ABB RobotStudio station: EstacionTaladrado.rspag

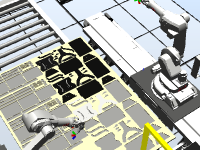
--- station ---
Station EstacionTaladrado (saved by RobotStudio 6.8.8307.1040)
Controller IRB1600APM, task T_ROB2: task frame (RAPID world) sits at (108, -1423.5, 460) mm, rotated rx 0 ry 0 rz 90 deg in the station
Controller IRB1600APM, task T_ROB1: task frame (RAPID world) sits at (108, -1423.5, 460) mm, rotated rx 0 ry 0 rz 90 deg in the station
Controller IRB1600APM
  mechanical unit ROB_1: IRB1600_6_145_A, 6 joints, base frame (0, 0, 0) mm
  mechanical unit TRACK_1: IRBT2005_IRB_STD_INT_0_0_4_A, 1 joints, base frame (0, 0, 0) mm
  mechanical unit ROB_2: IRB1600_6_145_B, 6 joints, base frame (1847, 2866, 0) mm, rotated rx 0 ry 0 rz 180 deg
  mechanical unit TRACK_2: IRBT2005_IRB_STD_INT_0_0_4_B, 1 joints, base frame (1847, 2866, 0) mm, rotated rx 0 ry 0 rz 180 deg
Layout (positions relative to the parent item):
  - Placa_de_Corte [part] at (-2250, -1220, 450) mm
  - IRC5_Singel-Cabinet [part, from Equipment\IRC5_Singel-Cabinet.rslib] at (500, 3000, 100) mm, rotated rx 90 ry 0 rz 90 deg
  - 1320_4000_h2 [part, from Equipment\Conveyor 1320 4000 h2.rslib] at (-1985, 2800, 0) mm, rotated rx 0 ry 0 rz -90 deg
  - Ventosa_Smart [smart component]
      signals: DI StartAttacher, DO Executed
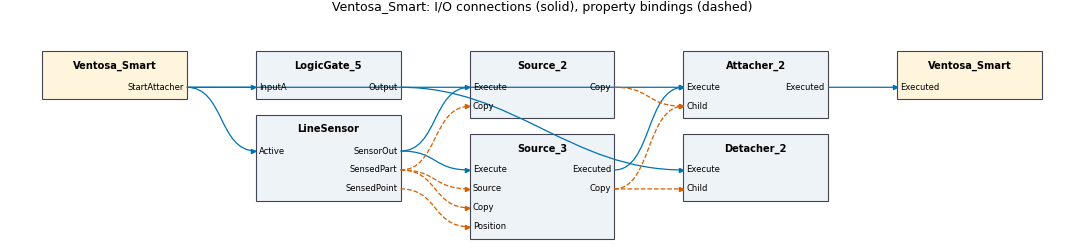
      connections:
        Ventosa_Smart.StartAttacher -> LogicGate_5.InputA
        LogicGate_5.Output -> Detacher_2.Execute
        Ventosa_Smart.StartAttacher -> LineSensor.Active
        Ventosa_Smart.StartAttacher -> Attacher_2.Execute
        Attacher_2.Executed -> Ventosa_Smart.Executed
        LineSensor.SensorOut -> Source_2.Execute
        LineSensor.SensorOut -> Source_3.Execute
        Source_3.Executed -> Attacher_2.Execute
        LineSensor.SensedPart => Source_2.Copy
        Source_2.Copy => Attacher_2.Child
        LineSensor.SensedPart => Source_3.Source
        LineSensor.SensedPart => Source_3.Copy
        Source_3.Copy => Attacher_2.Child
        Source_3.Copy => Detacher_2.Child
        LineSensor.SensedPoint => Source_3.Position
    - Attacher_2 [smart component, from Components\Attacher.rslib]
        properties: Parent=Ventosa; Flange=0; Child=(none); Mount=false; Offset=[0 0 0]; Orientation=[0 0 0]
    - Detacher_2 [smart component, from Components\Detacher.rslib]
        properties: Child=(none); KeepPosition=true
    - LogicGate_5 [smart component, from Components\LogicGate.rslib]
        properties: Operator=NOT; Delay=0
    - LineSensor [smart component, from Components\LineSensor.rslib] at (108, 403.05, 1559) mm, rotated rx 180 ry 60 rz -90 deg
        properties: Start=[0 0 0]; End=[6.66133814775094E-16 -4.71844785465692E-16 0.00999998807907376]; Radius=0.006; SensedPart=(none); SensedPoint=[0 0 0]
      - _sensorPart_ [part]
    - Ventosa [mechanism, from Libraries\Ventosa.rslib] at (108, 307.79, 1614) mm, rotated rx 180 ry 60 rz -90 deg
    - Source_3 [smart component, from Components\Source.rslib]
        properties: Source=(none); Copy=(none); Parent=(none); Position=[0 0 0]; Orientation=[0 0 0]; Transient=false; PhysicsBehavior=0
  - PLACA_SOPORTE_1 [part] at (-1200.46, 988.98, 450) mm
  - BANDEJA_LAMINA [part]
  - MyTool [mechanism, from Training Objects\myTool.rslib] at (-1542.16, -501.5, 845.83) mm, rotated rx 180 ry 0 rz 180 deg
  - SOPORTE_LATERAL_SOPORTE_1 [part] at (-961.81, 1075.54, 450) mm
  - MESA_TALADRADO [part] at (1200, -500, 400) mm
  - MESA_TALADRADO_B [part] at (-3850, -500, 400) mm
  - IRB1600_6_145_A [mechanism, from Robots\IRB1600_6_145_G_02.rslib] at (108, -498.5, 460) mm, rotated rx 0 ry 0 rz 90 deg; joint values [0, 0, 0, 0, 0.5236, 0] (rad or m)
  - IRB1600_6_145_B [mechanism, from Robots\IRB1600_6_145_G_02.rslib] at (-2758, -501.5, 460) mm, rotated rx 0 ry 0 rz -90 deg; joint values [1.5708, 1.0472, -0.3491, 0, 0.8727, 0] (rad or m)
  - IRBT2005_IRB_STD_INT_0_0_4_A [mechanism] at (400, -2248, 0) mm, rotated rx 0 ry 0 rz 90 deg; joint values [0.925] (rad or m)
      links: Base, Link1
  - IRBT2005_IRB_STD_INT_0_0_4_B [mechanism] at (-3050, 1248, 0) mm, rotated rx 0 ry 0 rz -90 deg; joint values [0.925] (rad or m)
      links: Base, Link1
  - Conveyor_A [smart component]
      signals: DI MoveConv
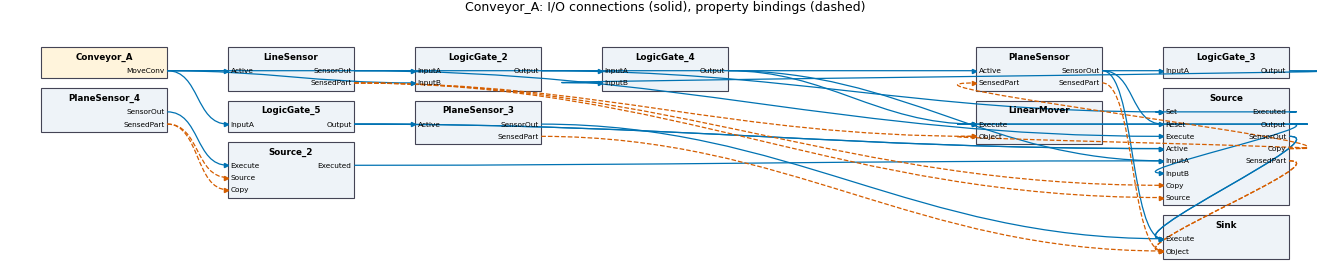
      connections:
        Source.Executed -> LogicSRLatch.Set
        PlaneSensor.SensorOut -> LogicSRLatch.Reset
        Conveyor_A.MoveConv -> LineSensor.Active
        LineSensor.SensorOut -> Source.Execute
        LogicSRLatch.Output -> LinearMover.Execute
        Conveyor_A.MoveConv -> PlaneSensor.Active
        LineSensor.SensorOut -> LogicGate_2.InputA
        Conveyor_A.MoveConv -> LogicGate_2.InputB
        LogicGate_2.Output -> LogicSRLatch.Set
        PlaneSensor.SensorOut -> LogicGate_3.InputA
        LogicGate_2.Output -> LogicGate_4.InputA
        LogicGate_3.Output -> LogicGate_4.InputB
        PlaneSensor.SensorOut -> Sink.Execute
        PlaneSensor_2.SensorOut -> Sink.Execute
        Conveyor_A.MoveConv -> LogicGate_5.InputA
        LogicGate_5.Output -> PlaneSensor_2.Active
        LogicGate_5.Output -> LineSensor.Active
        LineSensor.SensorOut -> Sink.Execute
        PlaneSensor_3.SensorOut -> Sink.Execute
        LogicGate_5.Output -> PlaneSensor_3.Active
        PlaneSensor_4.SensorOut -> Source_2.Execute
        LogicGate_4.Output -> LogicGate_8.InputA
        LogicGate_8.Output -> LinearMover.Execute
        LogicGate_9.Output -> LogicGate_8.InputB
        Source_2.Executed -> LogicGate_9.InputA
        LogicGate_4.Output -> LinearMover.Execute
        LineSensor.SensedPart => Source.Copy
        Source.Copy => LinearMover.Object
        Source.Copy => PlaneSensor.SensedPart
        LineSensor.SensedPart => Source.Source
        PlaneSensor_2.SensedPart => Sink.Object
        LineSensor.SensedPart => Sink.Object
        PlaneSensor_3.SensedPart => Sink.Object
        LineSensor.SensedPart => LinearMover.Object
        PlaneSensor.SensedPart => Sink.Object
        PlaneSensor_4.SensedPart => Source_2.Source
        PlaneSensor_4.SensedPart => Source_2.Copy
    - PlaneSensor [smart component, from Components\PlaneSensor.rslib]
        properties: Origin=[-1.025 -4.3 0.776]; Axis1=[0 0 0.099]; Axis2=[0.39 0 0]; SensedPart=(none)
      - _sensorPart_ [part]
    - LineSensor [smart component, from Components\LineSensor.rslib]
        properties: Start=[-0.83 -1.7 0.78]; End=[-0.83 -4.3 0.785]; Radius=0.005; SensedPart=BOX_A; SensedPoint=[-0.83 -1.7 0.78]
      - _sensorPart_ [part]
    - LinearMover [smart component, from Components\LinearMover.rslib]
        properties: Object=BOX_A; Direction=[0 -3.5 0]; Speed=0.5; Reference=Global; ReferenceObject=(none)
    - LogicGate_2 [smart component, from Components\LogicGate.rslib]
        properties: Operator=AND; Delay=0
    - LogicGate_3 [smart component, from Components\LogicGate.rslib]
        properties: Operator=NOT; Delay=0
    - LogicGate_4 [smart component, from Components\LogicGate.rslib]
        properties: Operator=AND; Delay=0
    - Sink [smart component, from Components\Sink.rslib]
        properties: Object=(none)
    - LogicGate_5 [smart component, from Components\LogicGate.rslib]
        properties: Operator=NOT; Delay=0
    - PlaneSensor_3 [smart component, from Components\PlaneSensor.rslib]
        properties: Origin=[-1.02 -2 0.786]; Axis1=[0.38 0 0]; Axis2=[0 0.3 0]; SensedPart=(none)
      - _sensorPart_ [part]
    - Source_2 [smart component, from Components\Source.rslib]
        properties: Source=(none); Copy=(none); Parent=(none); Position=[-0.83 -1.85 0.776]; Orientation=[0 0 0]; Transient=false; PhysicsBehavior=0
    - PlaneSensor_4 [smart component, from Components\PlaneSensor.rslib]
        properties: Origin=[-1.025 -4.3 0.776]; Axis1=[0 0 0.099]; Axis2=[0.39 0 0]; SensedPart=(none)
      - _sensorPart_ [part]
  - 400_guide_B [part, from Equipment\Conveyor Guide 400.rslib] at (-2020, -1500, 0) mm, rotated rx 0 ry 0 rz -90 deg
  - 400_guide_A [part, from Equipment\Conveyor Guide 400.rslib] at (-1030, -1500, 0) mm, rotated rx 0 ry 0 rz -90 deg
  - SOPORTE_LATERAL_SOPORTE_1_2 [part] at (-1011.44, 1038.99, 450) mm
  - BASE_SOPORTE_1 [part] at (-878.76, 996.15, 450) mm
  - GRADUADOR_INCLINACION_SOPORTE_1 [part] at (-1023.59, 997.95, 450) mm
  - GRADUADOR_INCLINACION_SOPORTE_1_2 [part] at (-966.4, 1160.33, 450) mm
  - SUJECION_CENTRAL_SOPORTE_1 [part] at (-870.47, 885.99, 450) mm
  - BRAZO_SOPORTE_1 [part] at (-762.24, 1077.84, 450) mm
  - BRAZO_2_SOPORTE_1 [part] at (-1135.46, 1150.12, 450) mm
  - BOX_A [part] at (-830, -1850, 776) mm
  - PLACA_INFERIOR_MESA_1 [part] at (-558.01, 1007.22, 450) mm
  - PLACA_SUPERIOR_MESA_1 [part] at (-913.92, 730.48, 450) mm
  - SOPORTE_LATERAL_I_MESA_1 [part] at (-1245.6, 782.8, 450) mm
  - SOPORTE_LATERAL_D_MESA_1 [part] at (-580.16, 719.3, 450) mm
  - BASE_SOPORTE_2 [part] at (-884.8, 433.69, 450) mm
  - BRAZO_2_SOPORTE_2 [part] at (-1248.93, 610.54, 450) mm
  - GRADUADOR_INCLINACION_SOPORTE_2 [part] at (-779.66, 491.03, 450) mm
  - GRADUADOR_INCLINACION_SOPORTE_2_2 [part] at (-777.34, 553.46, 450) mm
  - BRAZO_SOPORTE_3 [part] at (-1228.76, 84.41, 450) mm
  - BRAZO_SOPORTE_2 [part] at (-1242.31, 664.75, 450) mm
  - SOPORTE_LATERAL_SOPORTE_2 [part] at (-1012.51, 575.73, 450) mm
  - SOPORTE_LATERAL_SOPORTE_2_2 [part] at (-1009.84, 532.43, 450) mm
  - PLACA_SOPORTE_2 [part] at (-1204.37, 425.85, 450) mm
  - SUJECION_CENTRAL_SOPORTE_2 [part] at (-888.41, 308.37, 450) mm
  - PLACA_INFERIOR_MESA_2 [part] at (-580.45, 456.05, 450) mm
  - PLACA_SUPERIOR_MESA_2 [part] at (-915.16, 155.2, 450) mm
  - SOPORTE_LATERAL_I_MESA_2 [part] at (-1273.79, 206.85, 450) mm
  - SOPORTE_LATERAL_D_MESA_2 [part] at (-588.98, 160.74, 450) mm
  - BASE_SOPORTE_3 [part] at (-885, -169.85, 450) mm
  - PLACA_SOPORTE_3 [part] at (-1212.18, -176.73, 450) mm
  - Fence_2500 [graphiccomponentgroup, from Equipment\Fence_2500.rslib] at (-1350, -4000, 0) mm
    - Body 1 [part, from Equipment\Fence_2500.rslib]
    - Body 2 [part, from Equipment\Fence_2500.rslib]
  - Conveyor_B [smart component]
      signals: DI MoveConvB
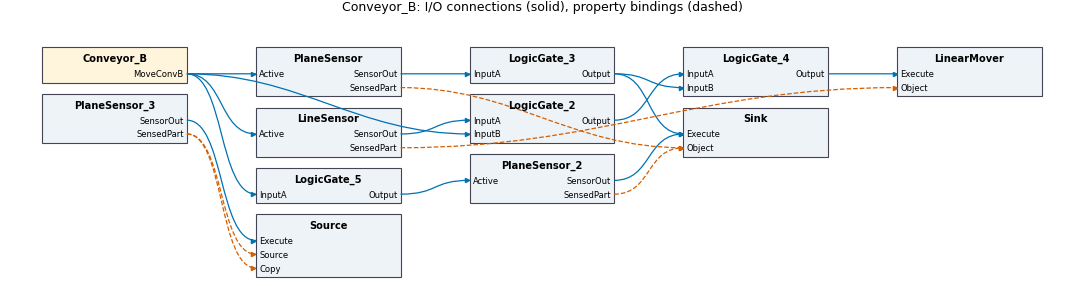
      connections:
        Conveyor_B.MoveConvB -> PlaneSensor.Active
        PlaneSensor.SensorOut -> LogicGate_3.InputA
        LogicGate_3.Output -> Sink.Execute
        Conveyor_B.MoveConvB -> LineSensor.Active
        LineSensor.SensorOut -> LogicGate_2.InputA
        Conveyor_B.MoveConvB -> LogicGate_5.InputA
        LogicGate_5.Output -> PlaneSensor_2.Active
        PlaneSensor_3.SensorOut -> Source.Execute
        LogicGate_2.Output -> LogicGate_4.InputA
        Conveyor_B.MoveConvB -> LogicGate_2.InputB
        LogicGate_3.Output -> LogicGate_4.InputB
        LogicGate_4.Output -> LinearMover.Execute
        PlaneSensor_2.SensorOut -> Sink.Execute
        PlaneSensor.SensedPart => Sink.Object
        LineSensor.SensedPart => LinearMover.Object
        PlaneSensor_3.SensedPart => Source.Source
        PlaneSensor_3.SensedPart => Source.Copy
        PlaneSensor_2.SensedPart => Sink.Object
    - LinearMover [smart component, from Components\LinearMover.rslib]
        properties: Object=BOX_A; Direction=[0 -3.5 0]; Speed=0.5; Reference=Global; ReferenceObject=(none)
    - LineSensor [smart component, from Components\LineSensor.rslib]
        properties: Start=[-1.82 -1.7 0.78]; End=[-1.82 -4.3 0.785]; Radius=0.005; SensedPart=BOX_A; SensedPoint=[-0.83 -1.7 0.78]
      - _sensorPart_ [part]
    - PlaneSensor [smart component, from Components\PlaneSensor.rslib]
        properties: Origin=[-2.02 -4.3 0.776]; Axis1=[0 0 0.099]; Axis2=[0.39 0 0]; SensedPart=(none)
      - _sensorPart_ [part]
    - PlaneSensor_2 [smart component, from Components\PlaneSensor.rslib]
        properties: Origin=[-2.01 -2 0.786]; Axis1=[0.38 0 0]; Axis2=[0 0.3 0]; SensedPart=(none)
      - _sensorPart_ [part]
    - PlaneSensor_3 [smart component, from Components\PlaneSensor.rslib]
        properties: Origin=[-2.02 -4.3 0.776]; Axis1=[0 0 0.099]; Axis2=[0.39 0 0]; SensedPart=(none)
      - _sensorPart_ [part]
    - Sink [smart component, from Components\Sink.rslib]
        properties: Object=(none)
    - Source [smart component, from Components\Source.rslib]
        properties: Source=(none); Copy=(none); Parent=(none); Position=[-0.83 -1.85 0.776]; Orientation=[0 0 0]; Transient=false; PhysicsBehavior=0
    - LogicGate_2 [smart component, from Components\LogicGate.rslib]
        properties: Operator=AND; Delay=0
    - LogicGate_3 [smart component, from Components\LogicGate.rslib]
        properties: Operator=NOT; Delay=0
    - LogicGate_4 [smart component, from Components\LogicGate.rslib]
        properties: Operator=AND; Delay=0
    - LogicGate_5 [smart component, from Components\LogicGate.rslib]
        properties: Operator=NOT; Delay=0
  - BOX_B [part] at (-1820, -1850, 776) mm
Attachment: LineSensor is attached to Ventosa / HERRAMIENTA
Attachment: Ventosa is attached to IRB1600_6_145_A / Link6
Attachment: MyTool is attached to IRB1600_6_145_B / Link6
Attachment: IRB1600_6_145_A is attached to IRBT2005_IRB_STD_INT_0_0_4_A / Link1
Attachment: IRB1600_6_145_B is attached to IRBT2005_IRB_STD_INT_0_0_4_B / Link1
Station logic (signal -> signal, property => property):
  Attacher.Executed -> LogicGate.InputB
  IRB1600APM.DOATTCH -> Ventosa_Smart.StartAttacher
  IRB1600APMSYS.DO_ATTCH_A -> Ventosa_Smart.StartAttacher
  IRB1600APM.ATTACH -> Ventosa_Smart.StartAttacher
  IRB1600APM.MoveConv -> Conveyor_A.MoveConv

--- Backups/IRB1600APM/RAPID/TASK1/PROGMOD/CalibData.mod ---
MODULE CalibData
	PERS tooldata VentosaTCP:=[TRUE,[[0,0,110.772],[1,0,0,0]],[1,[0,0,53.582],[1,0,0,0],0,0,0]];
	TASK PERS wobjdata PLACA_A:=[FALSE,TRUE,"",[[0,0,0],[1,0,0,0]],[[203.5,2358,-10],[0.707106781,0,0,-0.707106781]]];
ENDMODULE

--- Backups/IRB1600APM/RAPID/TASK1/PROGMOD/Module1.mod ---
MODULE Module1
    CONST jointtarget HOME_A:=[[0,0,0,0,30,0],[925,9E+09,9E+09,9E+09,9E+09,9E+09]];
    CONST jointtarget MID_A:=[[90,60,-20,0,50,0],[925,9E+09,9E+09,9E+09,9E+09,9E+09]];
    CONST jointtarget PS1_A:=[[87.22,84.052,-44.6,0,50.548,0],[2349.769019747,9E+09,9E+09,9E+09,9E+09,9E+09]];
    CONST jointtarget CONVEYOR_A:=[[84.914,41.92,15.328,-0.622,32.813,0],[-461.181385797,9E+09,9E+09,9E+09,9E+09,9E+09]];
    CONST jointtarget SLS1_A:=[[82.069,70.996,-7.558,0,26.562,-7.931],[2350,9E+09,9E+09,9E+09,9E+09,9E+09]];
    CONST jointtarget TABLE_A:=[[-90,71.536,-9.408,0,27.873,0],[925,9E+09,9E+09,9E+09,9E+09,9E+09]];
    CONST jointtarget PS1_AA:=[[87.22,83.446,-44.115,0,50.669,0],[2349.769019747,9E+09,9E+09,9E+09,9E+09,9E+09]];
    CONST jointtarget MID_CONV:=[[90,60,-40,0,70,0],[-500,9E+09,9E+09,9E+09,9E+09,9E+09]];
    CONST jointtarget MID_CONV_A:=[[89.175,20.381,4.444,0.004,65.253,0],[-480,9E+09,9E+09,9E+09,9E+09,9E+09]];
    CONST jointtarget PSLS1_AA:=[[82.069,69.527,-6.738,0,27.211,0],[2350,9E+09,9E+09,9E+09,9E+09,9E+09]];
    CONST jointtarget SLS12_AA:=[[84.262,72.054,-13.066,0,31.013,0],[2350,9E+09,9E+09,9E+09,9E+09,9E+09]];
    CONST jointtarget SLS12_A:=[[84.105,72.802,-13.543,0,30.74,-5.895],[2350,9E+09,9E+09,9E+09,9E+09,9E+09]];
    CONST jointtarget BS1_A:=[[84.635,68.196,3.223,0,18.581,0],[2350,9E+09,9E+09,9E+09,9E+09,9E+09]];
    CONST jointtarget BS1_AA:=[[84.635,67.383,3.658,0,18.96,0],[2350,9E+09,9E+09,9E+09,9E+09,9E+09]];
    CONST jointtarget GIS1_A:=[[86.51,72.86,-13.724,0,30.865,-3.49],[2350,9E+09,9E+09,9E+09,9E+09,9E+09]];
    CONST jointtarget GIS1_AA:=[[86.51,72.134,-13.296,0,31.162,0],[2350,9E+09,9E+09,9E+09,9E+09,9E+09]];
    CONST jointtarget GIS12_AA:=[[77.771,70.671,-8.671,0,28,0],[2350,9E+09,9E+09,9E+09,9E+09,9E+09]];
    CONST jointtarget GIS12_A:=[[77.79,71.449,-9.107,0,27.659,-12.21],[2350,9E+09,9E+09,9E+09,9E+09,9E+09]];
    CONST jointtarget BRS1_A:=[[80.135,66.069,14.969,0,8.962,-9.865],[2350,9E+09,9E+09,9E+09,9E+09,9E+09]];
    CONST jointtarget BRS1_AA:=[[80.135,65.237,15.395,0,9.368,0],[2350,9E+09,9E+09,9E+09,9E+09,9E+09]];
    CONST jointtarget BRS12_A:=[[79.805,80.411,-35.266,0,44.855,0],[2350,9E+09,9E+09,9E+09,9E+09,9E+09]];
    CONST jointtarget BRS12_AA:=[[79.805,79.69,-34.75,0,45.061,0],[2350,9E+09,9E+09,9E+09,9E+09,9E+09]];
    CONST jointtarget SCS1_A:=[[92.371,67.896,4.57,0,17.533,2.371],[2350,9E+09,9E+09,9E+09,9E+09,9E+09]];
    CONST jointtarget SCS1_AA:=[[92.371,67.108,4.99,0,17.903,0],[2350,9E+09,9E+09,9E+09,9E+09,9E+09]];
    CONST jointtarget PIM1_A:=[[56.022,65.432,22.991,0,1.578,-33.978],[1981.865508797,9E+09,9E+09,9E+09,9E+09,9E+09]];
    CONST jointtarget PIM1_AA:=[[56.022,64.534,23.445,0,2.021,-33.978],[1981.865508797,9E+09,9E+09,9E+09,9E+09,9E+09]];
    CONST jointtarget TABLE_AA:=[[-90,55.011,-3.204,0,38.193,0],[925,9E+09,9E+09,9E+09,9E+09,9E+09]];
    CONST jointtarget TABLE_A90:=[[-90.000002504,71.537536725,-9.40957169,0,27.872034908,90.000016165],[925.000071526,9E+09,9E+09,9E+09,9E+09,9E+09]];
    CONST jointtarget TABLE_A180:=[[-90,71.538,-9.41,0,27.872,180],[925.000071526,9E+09,9E+09,9E+09,9E+09,9E+09]];
    CONST jointtarget TABLE_A270:=[[-90,71.538,-9.41,0,27.872,270],[925.000071526,9E+09,9E+09,9E+09,9E+09,9E+09]];
    CONST jointtarget PSM1_AA:=[[80.44,68.736,-1.688,0.001,22.953,0],[1981.865508797,9E+09,9E+09,9E+09,9E+09,9E+09]];
    CONST jointtarget PSM1_A:=[[80.44,69.498,-2.107,0.001,22.609,0],[1981.865508797,9E+09,9E+09,9E+09,9E+09,9E+09]];
    CONST jointtarget SLIM1_AA:=[[80.586,90.25,-60.725,0,60.476,0],[1981.865508797,9E+09,9E+09,9E+09,9E+09,9E+09]];
    CONST jointtarget SLIM1_A:=[[80.586,91.085,-61.583,0,60.499,0],[1981.865508797,9E+09,9E+09,9E+09,9E+09,9E+09]];
    CONST jointtarget SLDM1_A:=[[76.838,65.923,31.968,-180,7.889,166.838],[1981.865508797,9E+09,9E+09,9E+09,9E+09,9E+09]];
    CONST jointtarget SLDM1_AA:=[[76.838,64.965,32.458,-180,7.42,166.838],[1981.865508797,9E+09,9E+09,9E+09,9E+09,9E+09]];
    CONST jointtarget SLS1_AA:=[[82.069,69.527,-6.738,0,27.211,0],[2350,9E+09,9E+09,9E+09,9E+09,9E+09]];
    CONST jointtarget TABLE_AA90:=[[-90,55.011,-3.204,0,38.193,90],[925,9E+09,9E+09,9E+09,9E+09,9E+09]];
    CONST jointtarget TABLE_AA180:=[[-90,55.011,-3.204,0,38.193,180],[925,9E+09,9E+09,9E+09,9E+09,9E+09]];
    CONST jointtarget TABLE_AA270:=[[-90,55.011,-3.204,0,38.193,270],[925,9E+09,9E+09,9E+09,9E+09,9E+09]];
    CONST jointtarget PS2_A:=[[92.202,84.352,-45.348,0,50.996,0],[1900.590004436,9E+09,9E+09,9E+09,9E+09,9E+09]];
    CONST jointtarget PS2_AA:=[[92.202,83.623,-44.761,0,51.138,0],[1900.590004436,9E+09,9E+09,9E+09,9E+09,9E+09]];
    CONST jointtarget BRS2_A:=[[82.088,89.838,-58.651,0,58.813,-7.912],[1900.590004436,9E+09,9E+09,9E+09,9E+09,9E+09]];
    CONST jointtarget BRS2_AA:=[[82.088,89.029,-57.86,0,58.831,-7.912],[1900.590004436,9E+09,9E+09,9E+09,9E+09,9E+09]];
    CONST jointtarget BRS22_A:=[[84.383,89.865,-58.714,0,58.849,0],[1900.590004436,9E+09,9E+09,9E+09,9E+09,9E+09]];
    CONST jointtarget BRS22_AA:=[[84.383,89.06,-57.926,0,58.866,0],[1900.590004436,9E+09,9E+09,9E+09,9E+09,9E+09]];
    CONST jointtarget BS2_A:=[[91.176,68.246,3.004,0,18.749,0],[1900.590004436,9E+09,9E+09,9E+09,9E+09,9E+09]];
    CONST jointtarget BS2_AA:=[[91.176,67.47,3.42,0,19.11,0],[1900.590004436,9E+09,9E+09,9E+09,9E+09,9E+09]];
    CONST jointtarget SLS2_A:=[[84.969,72.779,-13.468,0,30.689,-5.031],[1900.590004436,9E+09,9E+09,9E+09,9E+09,9E+09]];
    CONST jointtarget SLS2_AA:=[[84.969,72.056,-13.042,0,30.986,-5.031],[1900.590004436,9E+09,9E+09,9E+09,9E+09,9E+09]];
    CONST jointtarget SLS22_A:=[[87.166,72.539,-12.701,0,30.162,-2.834],[1900.590004436,9E+09,9E+09,9E+09,9E+09,9E+09]];
    CONST jointtarget SLS22_AA:=[[87.165999923,71.813298783,-12.275472962,-0.000004916,30.462172415,-2.833995324],[1900.590004436,9E+09,9E+09,9E+09,9E+09,9E+09]];
    CONST jointtarget GIS2_A:=[[113.168,67.339,7.247,0.002,15.415,23.166],[2350,9E+09,9E+09,9E+09,9E+09,9E+09]];
    CONST jointtarget GIS2_AA:=[[113.167997339,66.544675272,7.664479702,0.001953446,15.791846446,23.166056768],[2350,9E+09,9E+09,9E+09,9E+09,9E+09]];
    CONST jointtarget GIS22_A:=[[89.278,66.036,15.23,0,8.734,-0.722],[1900.590004436,9E+09,9E+09,9E+09,9E+09,9E+09]];
    CONST jointtarget GIS22_AA:=[[89.277996868,65.192591514,15.662153106,0,9.145254468,-0.722003182],[1900.590004436,9E+09,9E+09,9E+09,9E+09,9E+09]];
    CONST jointtarget SCS2_AA:=[[99.610427006,67.956188505,1.376250141,0.000001343,20.667561617,9.610424502],[1900.590004436,9E+09,9E+09,9E+09,9E+09,9E+09]];
    CONST jointtarget SCS2_A:=[[99.610427006,68.727863278,0.959277551,0.000002592,20.312857941,9.610423648],[1900.590004436,9E+09,9E+09,9E+09,9E+09,9E+09]];
    CONST jointtarget PIM2_AA:=[[91.561998466,65.215083327,34.070885788,-180.000005009,9.285968318,-178.437995387],[1898.318303054,9E+09,9E+09,9E+09,9E+09,9E+09]];
    CONST jointtarget PIM2_A:=[[91.562,66.191,33.57,-180,9.761,-178.438],[1898.318303054,9E+09,9E+09,9E+09,9E+09,9E+09]];
    CONST jointtarget PSM2_A:=[[107.463751193,70.721069572,-6.596925403,0,25.875854067,15.261750342],[1900.590004436,9E+09,9E+09,9E+09,9E+09,9E+09]];
    CONST jointtarget PSM2_AA:=[[107.463751193,69.981305443,-6.180146833,-0.000001709,26.198836637,15.261752049],[1900.590004436,9E+09,9E+09,9E+09,9E+09,9E+09]];
    CONST jointtarget SLIM2_AA:=[[101.065605639,97.834687105,-78.028074248,-0.000006825,70.193375987,8.863605642],[1900.590004436,9E+09,9E+09,9E+09,9E+09,9E+09]];
    CONST jointtarget SLIM2_A:=[[101.065605639,99.278479813,-80.225257312,-0.00000448,70.946766343,8.863604788],[1900.590004436,9E+09,9E+09,9E+09,9E+09,9E+09]];
    CONST jointtarget SLDM2_AA:=[[114.412894938,64.526784674,27.05293984,180.0003875,1.579731188,202.210537095],[1900.590004436,9E+09,9E+09,9E+09,9E+09,9E+09]];
    CONST jointtarget SLDM2_A:=[[114.412888108,65.445356325,26.587732241,179.999718141,2.033083713,202.211192794],[1900.590004436,9E+09,9E+09,9E+09,9E+09,9E+09]];
    !***********************************************************
    !
    ! Módulo:  Module1
    !
    ! Descripción:
    !   <Introduzca la descripción aquí>
    !
    ! Autor: sebas
    !
    ! Versión: 1.0
    !
    !***********************************************************


    !***********************************************************
    !
    ! Procedimiento Main
    !
    !   Este es el punto de entrada de su programa
    !
    !***********************************************************
    VAR intnum intparada;

    PROC main()
        !START
        CONNECT intparada WITH RutinaParada;
        iSignalDI STOPDI,1,intparada;
        SetDO MoveConv,0;
        WaitDI START,1;
        Path_HOME_A;
        Path_MID_A;
        !PLACA SOPORTE 1
        Path_PS1_AA;
        WaitTime 1;
        SetDO ATTACH,1;
        WaitDO ATTACH,1;
        Path_PS1_A;
        WaitTime 1;
        SetDO ATTACH,0;
        WaitDO ATTACH,0;
        Path_MID_CONV_A;
        Path_HOME_A;
        !SOPORTE LATERAL SOPORTE 1
        Path_SLS1_AA;
        WaitTime 1;
        SetDO ATTACH,1;
        WaitDO ATTACH,1;
        Path_SLS1_A;
        WaitDI DRILLCHECK,1;
        Path_SLS1_A_2;
        WaitTime 1;
        SetDO ATTACH,0;
        WaitDO ATTACH,0;
        Path_MID_CONV_A;
        Path_HOME_A;
        !SOPORTE LATERAL SOPORTE 1 2
        Path_SLS12_AA;
        WaitTime 1;
        SetDO ATTACH,1;
        WaitDO ATTACH,1;
        Path_SLS12_A;
        WaitDI DRILLCHECK,1;
        Path_SLS12_A_2;
        WaitTime 1;
        SetDO ATTACH,0;
        WaitDO ATTACH,0;
        Path_MID_CONV_A;
        Path_HOME_A;
        !BASE SOPORTE 1
        Path_BS1_AA;
        WaitTime 1;
        SetDO ATTACH,1;
        WaitDO ATTACH,1;
        Path_BS1_A;
        WaitTime 1;
        SetDO ATTACH,0;
        WaitDO ATTACH,0;
        Path_MID_CONV_A;
        Path_HOME_A;
        !GRADUADOR DE INCLINACION SOPORTE 1
        Path_GIS1_AA;
        WaitTime 1;
        SetDO ATTACH,1;
        WaitDO ATTACH,1;
        Path_GIS1_A;
        WaitDI DRILLCHECK,1;
        Path_GIS1_A_2;
        WaitTime 1;
        SetDO ATTACH,0;
        WaitDO ATTACH,0;
        Path_MID_CONV_A;
        Path_HOME_A;
        !GRADUADOR DE INCLINACION SOPORTE 1 2
        Path_GIS12_AA;
        WaitTime 1;
        SetDO ATTACH,1;
        WaitDO ATTACH,1;
        Path_GIS12_A;
        WaitDI DRILLCHECK,1;
        Path_GIS12_A_2;
        WaitTime 1;
        SetDO ATTACH,0;
        WaitDO ATTACH,0;
        Path_MID_CONV_A;
        Path_HOME_A;
        !BRAZO SOPORTE 1
        Path_BRS1_AA;
        WaitTime 1;
        SetDO ATTACH,1;
        WaitDO ATTACH,1;
        Path_BRS1_A;
        WaitTime 1;
        SetDO ATTACH,0;
        WaitDO ATTACH,0;
        Path_MID_CONV_A;
        Path_HOME_A;
        !BRAZO 2 SOPORTE 1
        Path_BRS12_AA;
        WaitTime 1;
        SetDO ATTACH,1;
        WaitDO ATTACH,1;
        Path_BRS12_A;
        WaitTime 1;
        SetDO ATTACH,0;
        WaitDO ATTACH,0;
        Path_MID_CONV_A;
        Path_HOME_A;
        !SUJECION CENTRAL SOPORTE 1
        Path_SCS1_AA;
        WaitTime 1;
        SetDO ATTACH,1;
        WaitDO ATTACH,1;
        Path_SCS1_A;
        WaitDI DRILLCHECK,1;
        Path_SCS1_A_2;
        WaitTime 1;
        SetDO ATTACH,0;
        WaitDO ATTACH,0;
        Path_MID_CONV_A;
        Path_HOME_A;
        !START CONVEYOR
        SetDO MoveConv,1;
        WaitTime 4.5;
        SetDO MoveConv,0;
        SetDO PAUSE,1;
        WaitDO PAUSE,0;
        !
        !MESA 1
        !
        !PLACA INFERIOR MESA 1
        Path_PIM1_AA;
        WaitTime 1;
        SetDO ATTACH,1;
        WaitDO ATTACH,1;
        Path_PIM1_A;
        WaitDI DRILLCHECK,1;
        WaitTime 1;
        Path_PIM1_A_2;
        WaitDI DRILLCHECK,1;
        WaitTime 1;
        Path_PIM1_A_3;
        WaitDI DRILLCHECK,1;
        WaitTime 1;
        Path_PIM1_A_4;
        WaitDI DRILLCHECK,1;
        WaitTime 1;
        Path_PIM1_A_5;
        WaitTime 1;
        SetDO ATTACH,0;
        WaitDO ATTACH,0;
        Path_MID_CONV_A;
        Path_HOME_A;
        !PLACA SUPERIOR MESA 1
        Path_PSM1_AA;
        WaitTime 1;
        SetDO ATTACH,1;
        WaitDO ATTACH,1;
        Path_PSM1_A;
        WaitTime 1;
        SetDO ATTACH,0;
        WaitDO ATTACH,0;
        Path_MID_CONV_A;
        Path_HOME_A;
        !SOPORTE LATERAL IZQUIERDO MESA 1
        Path_SLIM1_AA;
        WaitTime 1;
        SetDO ATTACH,1;
        WaitDO ATTACH,1;
        Path_SLIM1_A;
        WaitTime 1;
        SetDO ATTACH,0;
        WaitDO ATTACH,0;
        Path_MID_CONV_A;
        Path_HOME_A;
        !SOPORTE LATERAL DERECHO MESA 1
        Path_SLDM1_AA;
        WaitTime 1;
        SetDO ATTACH,1;
        WaitDO ATTACH,1;
        Path_SLDM1_A;
        WaitTime 1;
        SetDO ATTACH,0;
        WaitDO ATTACH,0;
        Path_MID_CONV_A;
        Path_HOME_A;
        !START CONVEYOR
        SetDO MoveConv,1;
        WaitTime 4.5;
        SetDO MoveConv,0;
        SetDO PAUSE,1;
        WaitDO PAUSE,0;
        !
        !SOPORTE 2
        !
        !PLACA SOPORTE 2
        Path_PS2_AA;
        WaitTime 1;
        SetDO ATTACH,1;
        WaitDO ATTACH,1;
        Path_PS2_A;
        WaitTime 1;
        SetDO ATTACH,0;
        WaitDO ATTACH,0;
        Path_MID_CONV_A;
        Path_HOME_A;
        !SOPORTE LATERAL SOPORTE 2
        Path_SLS2_AA;
        WaitTime 1;
        SetDO ATTACH,1;
        WaitDO ATTACH,1;
        Path_SLS2_A;
        WaitDI DRILLCHECK,1;
        Path_SLS2_A_2;
        WaitTime 1;
        SetDO ATTACH,0;
        WaitDO ATTACH,0;
        Path_MID_CONV_A;
        Path_HOME_A;
        !SOPORTE LATERAL SOPORTE 2 2
        Path_SLS22_AA;
        WaitTime 1;
        SetDO ATTACH,1;
        WaitDO ATTACH,1;
        Path_SLS22_A;
        WaitDI DRILLCHECK,1;
        Path_SLS22_A_2;
        WaitTime 1;
        SetDO ATTACH,0;
        WaitDO ATTACH,0;
        Path_MID_CONV_A;
        Path_HOME_A;
        !BASE SOPORTE 2
        Path_BS2_AA;
        WaitTime 1;
        SetDO ATTACH,1;
        WaitDO ATTACH,1;
        Path_BS2_A;
        WaitTime 1;
        SetDO ATTACH,0;
        WaitDO ATTACH,0;
        Path_MID_CONV_A;
        Path_HOME_A;
        !GRADUADOR DE INCLINACION SOPORTE 2
        Path_GIS2_AA;
        WaitTime 1;
        SetDO ATTACH,1;
        WaitDO ATTACH,1;
        Path_GIS2_A;
        WaitDI DRILLCHECK,1;
        Path_GIS2_A_2;
        WaitTime 1;
        SetDO ATTACH,0;
        WaitDO ATTACH,0;
        Path_MID_CONV_A;
        Path_HOME_A;
        !GRADUADOR DE INCLINACION SOPORTE 2 2
        Path_GIS22_AA;
        WaitTime 1;
        SetDO ATTACH,1;
        WaitDO ATTACH,1;
        Path_GIS22_A;
        WaitDI DRILLCHECK,1;
        Path_GIS22_A_2;
        WaitTime 1;
        SetDO ATTACH,0;
        WaitDO ATTACH,0;
        Path_MID_CONV_A;
        Path_HOME_A;
        !BRAZO SOPORTE 2
        Path_BRS2_AA;
        WaitTime 1;
        SetDO ATTACH,1;
        WaitDO ATTACH,1;
        Path_BRS2_A;
        WaitTime 1;
        SetDO ATTACH,0;
        WaitDO ATTACH,0;
        Path_MID_CONV_A;
        Path_HOME_A;
        !BRAZO 2 SOPORTE 2
        Path_BRS22_AA;
        WaitTime 1;
        SetDO ATTACH,1;
        WaitDO ATTACH,1;
        Path_BRS22_A;
        WaitTime 1;
        SetDO ATTACH,0;
        WaitDO ATTACH,0;
        Path_MID_CONV_A;
        Path_HOME_A;
        !SUJECION CENTRAL SOPORTE 2
        Path_SCS2_AA;
        WaitTime 1;
        SetDO ATTACH,1;
        WaitDO ATTACH,1;
        Path_SCS2_A;
        WaitDI DRILLCHECK,1;
        Path_SCS2_A_2;
        WaitTime 1;
        SetDO ATTACH,0;
        WaitDO ATTACH,0;
        Path_MID_CONV_A;
        Path_HOME_A;
        !START CONVEYOR
        SetDO MoveConv,1;
        WaitTime 4.5;
        SetDO MoveConv,0;
        SetDO PAUSE,1;
        WaitDO PAUSE,0;
        !
        !MESA 2
        !
        !PLACA INFERIOR MESA 2
        Path_PIM2_AA;
        WaitTime 1;
        SetDO ATTACH,1;
        WaitDO ATTACH,1;
        Path_PIM2_A;
        WaitDI DRILLCHECK,1;
        WaitTime 1;
        Path_PIM2_A_2;
        WaitDI DRILLCHECK,1;
        WaitTime 1;
        Path_PIM2_A_3;
        WaitDI DRILLCHECK,1;
        WaitTime 1;
        Path_PIM2_A_4;
        WaitDI DRILLCHECK,1;
        WaitTime 1;
        Path_PIM2_A_5;
        WaitTime 1;
        SetDO ATTACH,0;
        WaitDO ATTACH,0;
        Path_MID_CONV_A;
        Path_HOME_A;
        !PLACA SUPERIOR MESA 2
        Path_PSM2_AA;
        WaitTime 1;
        SetDO ATTACH,1;
        WaitDO ATTACH,1;
        Path_PSM2_A;
        WaitTime 1;
        SetDO ATTACH,0;
        WaitDO ATTACH,0;
        Path_MID_CONV_A;
        Path_HOME_A;
        !SOPORTE LATERAL IZQUIERDO MESA 2
        Path_SLIM2_AA;
        WaitTime 1;
        SetDO ATTACH,1;
        WaitDO ATTACH,1;
        Path_SLIM2_A;
        WaitTime 1;
        SetDO ATTACH,0;
        WaitDO ATTACH,0;
        Path_MID_CONV_A;
        Path_HOME_A;
        !SOPORTE LATERAL DERECHO MESA 2
        Path_SLDM2_AA;
        WaitTime 1;
        SetDO ATTACH,1;
        WaitDO ATTACH,1;
        Path_SLDM2_A;
        WaitTime 1;
        SetDO ATTACH,0;
        WaitDO ATTACH,0;
        Path_MID_CONV_A;
        Path_HOME_A;
        !START CONVEYOR
        SetDO MoveConv,1;
        WaitTime 4.5;
        SetDO MoveConv,0;
        SetDO PAUSE,1;
        WaitDO PAUSE,0;
        !
    ENDPROC

    TRAP RutinaParada
        StopMove;
        WaitDI STOPDI,0;
        StartMove;
    ENDTRAP

    PROC Path_HOME_A()
        MoveAbsJ HOME_A,v1500,z10,VentosaTCP\WObj:=PLACA_A;
    ENDPROC
    PROC Path_MID_A()
        MoveAbsJ MID_A,v1500,z10,VentosaTCP\WObj:=PLACA_A;
    ENDPROC
    PROC Path_S1_A()
        MoveAbsJ PS1_A,v1500,z10,VentosaTCP\WObj:=PLACA_A;
        MoveAbsJ MID_A,v1500,z10,VentosaTCP\WObj:=PLACA_A;
        MoveAbsJ CONVEYOR_A,v1500,z10,VentosaTCP\WObj:=PLACA_A;
    ENDPROC
    PROC Path_PS1_AA()
        MoveAbsJ PS1_AA,v1500,z10,VentosaTCP\WObj:=PLACA_A;
    ENDPROC
    PROC Path_PS1_A()
        MoveAbsJ PS1_A,v1500,z10,VentosaTCP\WObj:=PLACA_A;
        MoveAbsJ PS1_AA,v1500,z10,VentosaTCP\WObj:=PLACA_A;
        MoveAbsJ HOME_A,v1500,z10,VentosaTCP\WObj:=PLACA_A;
        MoveAbsJ MID_CONV_A,v1500,z10,VentosaTCP\WObj:=PLACA_A;
        MoveAbsJ CONVEYOR_A,v1500,z10,VentosaTCP\WObj:=PLACA_A;
    ENDPROC
    PROC Path_MID_CONV_A()
        MoveAbsJ MID_CONV_A,v1500,z10,VentosaTCP\WObj:=PLACA_A;
    ENDPROC
    PROC Path_SLS1_A()
        MoveAbsJ SLS1_A,v1500,z10,VentosaTCP\WObj:=PLACA_A;
        MoveAbsJ SLS1_AA,v1500,z10,VentosaTCP\WObj:=PLACA_A;
        MoveAbsJ MID_A,v1500,z10,VentosaTCP\WObj:=PLACA_A;
        MoveAbsJ HOME_A,v1500,z10,VentosaTCP\WObj:=PLACA_A;
        MoveAbsJ TABLE_AA,v1500,z10,VentosaTCP\WObj:=PLACA_A;
        MoveAbsJ TABLE_A,v1500,z10,VentosaTCP\WObj:=PLACA_A;
    ENDPROC
    PROC Path_SLS1_AA()
        MoveAbsJ SLS1_AA,v1500,z10,VentosaTCP\WObj:=PLACA_A;
    ENDPROC
    PROC Path_SLS12_AA()
        MoveAbsJ SLS12_AA,v1500,z10,VentosaTCP\WObj:=PLACA_A;
    ENDPROC
    PROC Path_SLS12_A()
        MoveAbsJ SLS12_A,v1500,z10,VentosaTCP\WObj:=PLACA_A;
        MoveAbsJ SLS12_AA,v1500,z10,VentosaTCP\WObj:=PLACA_A;
        MoveAbsJ MID_A,v1500,z10,VentosaTCP\WObj:=PLACA_A;
        MoveAbsJ HOME_A,v1500,z10,VentosaTCP\WObj:=PLACA_A;
        MoveAbsJ TABLE_A,v1500,z10,VentosaTCP\WObj:=PLACA_A;
    ENDPROC
    PROC Path_BS1_A()
        MoveAbsJ BS1_A,v1500,z10,VentosaTCP\WObj:=PLACA_A;
        MoveAbsJ BS1_AA,v1500,z10,VentosaTCP\WObj:=PLACA_A;
        MoveAbsJ MID_A,v1500,z10,VentosaTCP\WObj:=PLACA_A;
        MoveAbsJ HOME_A,v1500,z10,VentosaTCP\WObj:=PLACA_A;
        MoveAbsJ MID_CONV_A,v1500,z10,VentosaTCP\WObj:=PLACA_A;
        MoveAbsJ CONVEYOR_A,v1500,z10,VentosaTCP\WObj:=PLACA_A;
    ENDPROC
    PROC Path_BS1_AA()
        MoveAbsJ BS1_AA,v1500,z10,VentosaTCP\WObj:=PLACA_A;
    ENDPROC
    PROC Path_SLS1_A_2()
        MoveAbsJ HOME_A,v1500,z10,VentosaTCP\WObj:=PLACA_A;
        MoveAbsJ MID_CONV_A,v1500,z10,VentosaTCP\WObj:=PLACA_A;
        MoveAbsJ CONVEYOR_A,v1500,z10,VentosaTCP\WObj:=PLACA_A;
    ENDPROC
    PROC Path_SLS12_A_2()
        MoveAbsJ HOME_A,v1500,z10,VentosaTCP\WObj:=PLACA_A;
        MoveAbsJ MID_CONV_A,v1500,z10,VentosaTCP\WObj:=PLACA_A;
        MoveAbsJ CONVEYOR_A,v1500,z10,VentosaTCP\WObj:=PLACA_A;
    ENDPROC
    PROC Path_GIS1_A()
        MoveAbsJ GIS1_A,v1500,z10,VentosaTCP\WObj:=PLACA_A;
        MoveAbsJ GIS1_AA,v1500,z10,VentosaTCP\WObj:=PLACA_A;
        MoveAbsJ MID_A,v1500,z10,VentosaTCP\WObj:=PLACA_A;
        MoveAbsJ HOME_A,v1500,z10,VentosaTCP\WObj:=PLACA_A;
        MoveAbsJ TABLE_A,v1500,z10,VentosaTCP\WObj:=PLACA_A;

    ENDPROC
    PROC Path_GIS1_AA()
        MoveAbsJ GIS1_AA,v1500,z10,VentosaTCP\WObj:=PLACA_A;
    ENDPROC
    PROC Path_GIS1_A_2()
        MoveAbsJ TABLE_AA,v1500,z10,VentosaTCP\WObj:=PLACA_A;
        MoveAbsJ HOME_A,v1500,z10,VentosaTCP\WObj:=PLACA_A;
        MoveAbsJ MID_CONV_A,v1500,z10,VentosaTCP\WObj:=PLACA_A;
        MoveAbsJ CONVEYOR_A,v1500,z10,VentosaTCP\WObj:=PLACA_A;
    ENDPROC
    PROC Path_GIS12_AA()
        MoveAbsJ GIS12_AA,v1500,z10,VentosaTCP\WObj:=PLACA_A;
    ENDPROC
    PROC Path_GIS12_A()
        MoveAbsJ GIS12_A,v1500,z10,VentosaTCP\WObj:=PLACA_A;
        MoveAbsJ GIS12_AA,v1500,z10,VentosaTCP\WObj:=PLACA_A;
        MoveAbsJ MID_A,v1500,z10,VentosaTCP\WObj:=PLACA_A;
        MoveAbsJ HOME_A,v1500,z10,VentosaTCP\WObj:=PLACA_A;
        MoveAbsJ TABLE_A,v1500,z10,VentosaTCP\WObj:=PLACA_A;
    ENDPROC
    PROC Path_GIS12_A_2()
        MoveAbsJ HOME_A,v1500,z10,VentosaTCP\WObj:=PLACA_A;
        MoveAbsJ MID_CONV_A,v1500,z10,VentosaTCP\WObj:=PLACA_A;
        MoveAbsJ CONVEYOR_A,v1500,z10,VentosaTCP\WObj:=PLACA_A;
    ENDPROC
    PROC Path_BRS1_A()
        MoveAbsJ BRS1_A,v1500,z10,VentosaTCP\WObj:=PLACA_A;
        MoveAbsJ BRS1_AA,v1500,z10,VentosaTCP\WObj:=PLACA_A;
        MoveAbsJ MID_A,v1500,z10,VentosaTCP\WObj:=PLACA_A;
        MoveAbsJ HOME_A,v1500,z10,VentosaTCP\WObj:=PLACA_A;
        MoveAbsJ MID_CONV_A,v1500,z10,VentosaTCP\WObj:=PLACA_A;
        MoveAbsJ CONVEYOR_A,v1500,z10,VentosaTCP\WObj:=PLACA_A;
    ENDPROC
    PROC Path_BRS1_AA()
        MoveAbsJ BRS1_AA,v1500,z10,VentosaTCP\WObj:=PLACA_A;
    ENDPROC
    PROC Path_BRS12_A()
        MoveAbsJ BRS12_A,v1500,z10,VentosaTCP\WObj:=PLACA_A;
        MoveAbsJ BRS12_AA,v1500,z10,VentosaTCP\WObj:=PLACA_A;
        MoveAbsJ MID_A,v1500,z10,VentosaTCP\WObj:=PLACA_A;
        MoveAbsJ HOME_A,v1500,z10,VentosaTCP\WObj:=PLACA_A;
        MoveAbsJ MID_CONV_A,v1500,z10,VentosaTCP\WObj:=PLACA_A;
        MoveAbsJ CONVEYOR_A,v1500,z10,VentosaTCP\WObj:=PLACA_A;
    ENDPROC
    PROC Path_BRS12_AA()
        MoveAbsJ BRS12_AA,v1500,z10,VentosaTCP\WObj:=PLACA_A;
    ENDPROC
    PROC Path_SCS1_A()
        MoveAbsJ SCS1_A,v1500,z10,VentosaTCP\WObj:=PLACA_A;
        MoveAbsJ SCS1_AA,v1500,z10,VentosaTCP\WObj:=PLACA_A;
        MoveAbsJ MID_A,v1500,z10,VentosaTCP\WObj:=PLACA_A;
        MoveAbsJ HOME_A,v1500,z10,VentosaTCP\WObj:=PLACA_A;
        MoveAbsJ TABLE_A,v1500,z10,VentosaTCP\WObj:=PLACA_A;
    ENDPROC
    PROC Path_SCS1_AA()
        MoveAbsJ SCS1_AA,v1500,z10,VentosaTCP\WObj:=PLACA_A;
    ENDPROC
    PROC Path_SCS1_A_2()
        MoveAbsJ HOME_A,v1500,z10,VentosaTCP\WObj:=PLACA_A;
        MoveAbsJ MID_CONV_A,v1500,z10,VentosaTCP\WObj:=PLACA_A;
        MoveAbsJ CONVEYOR_A,v1500,z10,VentosaTCP\WObj:=PLACA_A;
    ENDPROC
    PROC Path_PIM1_A()
        MoveAbsJ PIM1_A,v1500,z10,VentosaTCP\WObj:=PLACA_A;
        MoveAbsJ PIM1_AA,v1500,z10,VentosaTCP\WObj:=PLACA_A;
        MoveAbsJ MID_A,v1500,z10,VentosaTCP\WObj:=PLACA_A;
        MoveAbsJ HOME_A,v1500,z10,VentosaTCP\WObj:=PLACA_A;
        MoveAbsJ TABLE_AA,v1500,z10,VentosaTCP\WObj:=PLACA_A;
        MoveAbsJ TABLE_A,v1500,z10,VentosaTCP\WObj:=PLACA_A;
    ENDPROC
    PROC Path_PIM1_AA()
        MoveAbsJ PIM1_AA,v1500,z10,VentosaTCP\WObj:=PLACA_A;
    ENDPROC
    PROC Path_PIM1_A_2()
        MoveAbsJ TABLE_AA90,v1500,z10,VentosaTCP\WObj:=PLACA_A;
        MoveAbsJ TABLE_A90,v1500,z10,VentosaTCP\WObj:=PLACA_A;
    ENDPROC
    PROC Path_PIM1_A_3()
        MoveAbsJ TABLE_AA180,v1500,z10,VentosaTCP\WObj:=PLACA_A;
        MoveAbsJ TABLE_A180,v1500,z10,VentosaTCP\WObj:=PLACA_A;
    ENDPROC
    PROC Path_PIM1_A_4()
        MoveAbsJ TABLE_AA270,v1500,z10,VentosaTCP\WObj:=PLACA_A;
        MoveAbsJ TABLE_A270,v1500,z10,VentosaTCP\WObj:=PLACA_A;
    ENDPROC
    PROC Path_PIM1_A_5()
        MoveAbsJ TABLE_AA,v1500,z10,VentosaTCP\WObj:=PLACA_A;
        MoveAbsJ HOME_A,v1500,z10,VentosaTCP\WObj:=PLACA_A;
        MoveAbsJ MID_CONV_A,v1500,z10,VentosaTCP\WObj:=PLACA_A;
        MoveAbsJ CONVEYOR_A,v1500,z10,VentosaTCP\WObj:=PLACA_A;
    ENDPROC
    PROC Path_PSM1_AA()
        MoveAbsJ PSM1_AA,v1500,z10,VentosaTCP\WObj:=PLACA_A;
    ENDPROC
    PROC Path_PSM1_A()
        MoveAbsJ PSM1_A,v1500,z10,VentosaTCP\WObj:=PLACA_A;
        MoveAbsJ PSM1_AA,v1500,z10,VentosaTCP\WObj:=PLACA_A;
        MoveAbsJ MID_A,v1500,z10,VentosaTCP\WObj:=PLACA_A;
        MoveAbsJ HOME_A,v1500,z10,VentosaTCP\WObj:=PLACA_A;
        MoveAbsJ MID_CONV_A,v1500,z10,VentosaTCP\WObj:=PLACA_A;
        MoveAbsJ CONVEYOR_A,v1500,z10,VentosaTCP\WObj:=PLACA_A;
    ENDPROC
    PROC Path_SLIM1_AA()
        MoveAbsJ SLIM1_AA,v1500,z10,VentosaTCP\WObj:=PLACA_A;
    ENDPROC
    PROC Path_SLIM1_A()
        MoveAbsJ SLIM1_A,v1500,z10,VentosaTCP\WObj:=PLACA_A;
        MoveAbsJ SLIM1_AA,v1500,z10,VentosaTCP\WObj:=PLACA_A;
        MoveAbsJ MID_A,v1500,z10,VentosaTCP\WObj:=PLACA_A;
        MoveAbsJ HOME_A,v1500,z10,VentosaTCP\WObj:=PLACA_A;
        MoveAbsJ MID_CONV_A,v1500,z10,VentosaTCP\WObj:=PLACA_A;
        MoveAbsJ CONVEYOR_A,v1500,z10,VentosaTCP\WObj:=PLACA_A;
    ENDPROC
    PROC Path_SLDM1_A()
        MoveAbsJ SLDM1_A,v1500,z10,VentosaTCP\WObj:=PLACA_A;
        MoveAbsJ SLDM1_AA,v1500,z10,VentosaTCP\WObj:=PLACA_A;
        MoveAbsJ MID_A,v1500,z10,VentosaTCP\WObj:=PLACA_A;
        MoveAbsJ HOME_A,v1500,z10,VentosaTCP\WObj:=PLACA_A;
        MoveAbsJ MID_CONV_A,v1500,z10,VentosaTCP\WObj:=PLACA_A;
        MoveAbsJ CONVEYOR_A,v1500,z10,VentosaTCP\WObj:=PLACA_A;
    ENDPROC
    PROC Path_SLDM1_AA()
        MoveAbsJ SLDM1_AA,v1500,z10,VentosaTCP\WObj:=PLACA_A;
    ENDPROC
    PROC Path_PS2_A()
        MoveAbsJ PS2_A,v1500,z10,VentosaTCP\WObj:=PLACA_A;
        MoveAbsJ PS2_AA,v1500,z10,VentosaTCP\WObj:=PLACA_A;
        MoveAbsJ MID_A,v1500,z10,VentosaTCP\WObj:=PLACA_A;
        MoveAbsJ HOME_A,v1500,z10,VentosaTCP\WObj:=PLACA_A;
        MoveAbsJ MID_CONV_A,v1500,z10,VentosaTCP\WObj:=PLACA_A;
        MoveAbsJ CONVEYOR_A,v1500,z10,VentosaTCP\WObj:=PLACA_A;
    ENDPROC
    PROC Path_PS2_AA()
        MoveAbsJ PS2_AA,v1500,z10,VentosaTCP\WObj:=PLACA_A;
    ENDPROC
    PROC Path_BRS2_A()
        MoveAbsJ BRS2_A,v1500,z10,VentosaTCP\WObj:=PLACA_A;
        MoveAbsJ BRS2_AA,v1500,z10,VentosaTCP\WObj:=PLACA_A;
        MoveAbsJ MID_A,v1500,z10,VentosaTCP\WObj:=PLACA_A;
        MoveAbsJ HOME_A,v1500,z10,VentosaTCP\WObj:=PLACA_A;
        MoveAbsJ MID_CONV_A,v1500,z10,VentosaTCP\WObj:=PLACA_A;
        MoveAbsJ CONVEYOR_A,v1500,z10,VentosaTCP\WObj:=PLACA_A;
    ENDPROC
    PROC Path_BRS2_AA()
        MoveAbsJ BRS2_AA,v1500,z10,VentosaTCP\WObj:=PLACA_A;
    ENDPROC
    PROC Path_BRS22_A()
        MoveAbsJ BRS22_A,v1500,z10,VentosaTCP\WObj:=PLACA_A;
        MoveAbsJ BRS22_AA,v1500,z10,VentosaTCP\WObj:=PLACA_A;
        MoveAbsJ MID_A,v1500,z10,VentosaTCP\WObj:=PLACA_A;
        MoveAbsJ HOME_A,v1500,z10,VentosaTCP\WObj:=PLACA_A;
        MoveAbsJ MID_CONV_A,v1500,z10,VentosaTCP\WObj:=PLACA_A;
        MoveAbsJ CONVEYOR_A,v1500,z10,VentosaTCP\WObj:=PLACA_A;
    ENDPROC
    PROC Path_BRS22_AA()
        MoveAbsJ BRS22_AA,v1500,z10,VentosaTCP\WObj:=PLACA_A;
    ENDPROC
    PROC Path_BS2_A()
        MoveAbsJ BS2_A,v1500,z10,VentosaTCP\WObj:=PLACA_A;
        MoveAbsJ BS2_AA,v1500,z10,VentosaTCP\WObj:=PLACA_A;
        MoveAbsJ MID_A,v1500,z10,VentosaTCP\WObj:=PLACA_A;
        MoveAbsJ HOME_A,v1500,z10,VentosaTCP\WObj:=PLACA_A;
        MoveAbsJ MID_CONV_A,v1500,z10,VentosaTCP\WObj:=PLACA_A;
        MoveAbsJ CONVEYOR_A,v1500,z10,VentosaTCP\WObj:=PLACA_A;
    ENDPROC
    PROC Path_BS2_AA()
        MoveAbsJ BS2_AA,v1500,z10,VentosaTCP\WObj:=PLACA_A;
    ENDPROC
    PROC Path_SLS2_A()
        MoveAbsJ SLS2_A,v1500,z10,VentosaTCP\WObj:=PLACA_A;
        MoveAbsJ SLS2_AA,v1500,z10,VentosaTCP\WObj:=PLACA_A;
        MoveAbsJ MID_A,v1500,z10,VentosaTCP\WObj:=PLACA_A;
        MoveAbsJ HOME_A,v1500,z10,VentosaTCP\WObj:=PLACA_A;
        MoveAbsJ TABLE_AA,v1500,z10,VentosaTCP\WObj:=PLACA_A;
        MoveAbsJ TABLE_A,v1500,z10,VentosaTCP\WObj:=PLACA_A;
    ENDPROC
    PROC Path_SLS2_AA()
        MoveAbsJ SLS2_AA,v1500,z10,VentosaTCP\WObj:=PLACA_A;
    ENDPROC
    PROC Path_SLS2_A_2()
        MoveAbsJ TABLE_AA,v1500,z10,VentosaTCP\WObj:=PLACA_A;
        MoveAbsJ HOME_A,v1500,z10,VentosaTCP\WObj:=PLACA_A;
        MoveAbsJ MID_CONV_A,v1500,z10,VentosaTCP\WObj:=PLACA_A;
        MoveAbsJ CONVEYOR_A,v1500,z10,VentosaTCP\WObj:=PLACA_A;
    ENDPROC
    PROC Path_SLS22_A()
        MoveAbsJ SLS22_A,v1500,z10,VentosaTCP\WObj:=PLACA_A;
        MoveAbsJ SLS22_AA,v1500,z10,VentosaTCP\WObj:=PLACA_A;
        MoveAbsJ MID_A,v1500,z10,VentosaTCP\WObj:=PLACA_A;
        MoveAbsJ HOME_A,v1500,z10,VentosaTCP\WObj:=PLACA_A;
        MoveAbsJ TABLE_AA,v1500,z10,VentosaTCP\WObj:=PLACA_A;
        MoveAbsJ TABLE_A,v1500,z10,VentosaTCP\WObj:=PLACA_A;
    ENDPROC
    PROC Path_SLS22_AA()
        MoveAbsJ SLS22_AA,v1500,z10,VentosaTCP\WObj:=PLACA_A;
    ENDPROC
    PROC Path_SLS22_A_2()
        MoveAbsJ TABLE_AA,v1500,z10,VentosaTCP\WObj:=PLACA_A;
        MoveAbsJ HOME_A,v1500,z10,VentosaTCP\WObj:=PLACA_A;
        MoveAbsJ MID_CONV_A,v1500,z10,VentosaTCP\WObj:=PLACA_A;
        MoveAbsJ CONVEYOR_A,v1500,z10,VentosaTCP\WObj:=PLACA_A;
    ENDPROC
    PROC Path_GIS2_A()
        MoveAbsJ GIS2_A,v1500,z10,VentosaTCP\WObj:=PLACA_A;
        MoveAbsJ GIS2_AA,v1500,z10,VentosaTCP\WObj:=PLACA_A;
        MoveAbsJ MID_A,v1500,z10,VentosaTCP\WObj:=PLACA_A;
        MoveAbsJ HOME_A,v1500,z10,VentosaTCP\WObj:=PLACA_A;
        MoveAbsJ TABLE_A,v1500,z10,VentosaTCP\WObj:=PLACA_A;
    ENDPROC
    PROC Path_GIS2_A_2()
        MoveAbsJ TABLE_AA,v1500,z10,VentosaTCP\WObj:=PLACA_A;
        MoveAbsJ HOME_A,v1500,z10,VentosaTCP\WObj:=PLACA_A;
        MoveAbsJ MID_CONV_A,v1500,z10,VentosaTCP\WObj:=PLACA_A;
        MoveAbsJ CONVEYOR_A,v1500,z10,VentosaTCP\WObj:=PLACA_A;
    ENDPROC
    PROC Path_GIS2_AA()
        MoveAbsJ GIS2_AA,v1500,z10,VentosaTCP\WObj:=PLACA_A;
    ENDPROC
    PROC Path_GIS2_A_3()
        MoveAbsJ GIS2_A,v1500,z10,VentosaTCP\WObj:=PLACA_A;
        MoveAbsJ GIS2_AA,v1500,z10,VentosaTCP\WObj:=PLACA_A;
        MoveAbsJ MID_A,v1500,z10,VentosaTCP\WObj:=PLACA_A;
        MoveAbsJ HOME_A,v1500,z10,VentosaTCP\WObj:=PLACA_A;
        MoveAbsJ TABLE_A,v1500,z10,VentosaTCP\WObj:=PLACA_A;
    ENDPROC
    PROC Path_GIS2_A_2_2()
        MoveAbsJ TABLE_AA,v1500,z10,VentosaTCP\WObj:=PLACA_A;
        MoveAbsJ HOME_A,v1500,z10,VentosaTCP\WObj:=PLACA_A;
        MoveAbsJ MID_CONV_A,v1500,z10,VentosaTCP\WObj:=PLACA_A;
        MoveAbsJ CONVEYOR_A,v1500,z10,VentosaTCP\WObj:=PLACA_A;
    ENDPROC
    PROC Path_GIS2_AA_2()
        MoveAbsJ GIS2_AA,v1500,z10,VentosaTCP\WObj:=PLACA_A;
    ENDPROC
    PROC Path_GIS22_A()
        MoveAbsJ GIS22_A,v1500,z10,VentosaTCP\WObj:=PLACA_A;
        MoveAbsJ GIS22_AA,v1500,z10,VentosaTCP\WObj:=PLACA_A;
        MoveAbsJ MID_A,v1500,z10,VentosaTCP\WObj:=PLACA_A;
        MoveAbsJ HOME_A,v1500,z10,VentosaTCP\WObj:=PLACA_A;
        MoveAbsJ TABLE_A,v1500,z10,VentosaTCP\WObj:=PLACA_A;
    ENDPROC
    PROC Path_GIS22_A_2()
        MoveAbsJ TABLE_AA,v1500,z10,VentosaTCP\WObj:=PLACA_A;
        MoveAbsJ HOME_A,v1500,z10,VentosaTCP\WObj:=PLACA_A;
        MoveAbsJ MID_CONV_A,v1500,z10,VentosaTCP\WObj:=PLACA_A;
        MoveAbsJ CONVEYOR_A,v1500,z10,VentosaTCP\WObj:=PLACA_A;
    ENDPROC
    PROC Path_GIS22_AA()
        MoveAbsJ GIS22_AA,v1500,z10,VentosaTCP\WObj:=PLACA_A;
    ENDPROC
    PROC Path_SCS2_AA()
        MoveAbsJ SCS2_AA,v1500,z10,VentosaTCP\WObj:=PLACA_A;
    ENDPROC
    PROC Path_SCS2_A()
        MoveAbsJ SCS2_A,v1500,z10,VentosaTCP\WObj:=PLACA_A;
        MoveAbsJ SCS2_AA,v1500,z10,VentosaTCP\WObj:=PLACA_A;
        MoveAbsJ MID_A,v1500,z10,VentosaTCP\WObj:=PLACA_A;
        MoveAbsJ HOME_A,v1500,z10,VentosaTCP\WObj:=PLACA_A;
        MoveAbsJ TABLE_AA,v1500,z10,VentosaTCP\WObj:=PLACA_A;
        MoveAbsJ TABLE_A,v1500,z10,VentosaTCP\WObj:=PLACA_A;
    ENDPROC
    PROC Path_SCS2_A_2()
        MoveAbsJ TABLE_AA,v1500,z10,VentosaTCP\WObj:=PLACA_A;
        MoveAbsJ HOME_A,v1500,z10,VentosaTCP\WObj:=PLACA_A;
        MoveAbsJ MID_CONV_A,v1500,z10,VentosaTCP\WObj:=PLACA_A;
        MoveAbsJ CONVEYOR_A,v1500,z10,VentosaTCP\WObj:=PLACA_A;
    ENDPROC
    PROC Path_PIM2_AA()
        MoveAbsJ PIM2_AA,v1500,z10,VentosaTCP\WObj:=PLACA_A;
    ENDPROC
    PROC Path_PIM2_A()
        MoveAbsJ PIM2_A,v1500,z10,VentosaTCP\WObj:=PLACA_A;
        MoveAbsJ PIM2_AA,v1500,z10,VentosaTCP\WObj:=PLACA_A;
        MoveAbsJ MID_A,v1500,z10,VentosaTCP\WObj:=PLACA_A;
        MoveAbsJ HOME_A,v1500,z10,VentosaTCP\WObj:=PLACA_A;
        MoveAbsJ TABLE_AA,v1500,z10,VentosaTCP\WObj:=PLACA_A;
        MoveAbsJ TABLE_A,v1500,z10,VentosaTCP\WObj:=PLACA_A;
    ENDPROC
    PROC Path_PIM2_A_2()
        MoveAbsJ TABLE_AA90,v1500,z10,VentosaTCP\WObj:=PLACA_A;
        MoveAbsJ TABLE_A90,v1500,z10,VentosaTCP\WObj:=PLACA_A;
    ENDPROC
    PROC Path_PIM2_A_3()
        MoveAbsJ TABLE_AA180,v1500,z10,VentosaTCP\WObj:=PLACA_A;
        MoveAbsJ TABLE_A180,v1500,z10,VentosaTCP\WObj:=PLACA_A;
    ENDPROC
    PROC Path_PIM2_A_4()
        MoveAbsJ TABLE_AA270,v1500,z10,VentosaTCP\WObj:=PLACA_A;
        MoveAbsJ TABLE_A270,v1500,z10,VentosaTCP\WObj:=PLACA_A;
    ENDPROC
    PROC Path_PIM2_A_5()
        MoveAbsJ TABLE_AA,v1500,z10,VentosaTCP\WObj:=PLACA_A;
        MoveAbsJ HOME_A,v1500,z10,VentosaTCP\WObj:=PLACA_A;
        MoveAbsJ MID_CONV_A,v1500,z10,VentosaTCP\WObj:=PLACA_A;
        MoveAbsJ CONVEYOR_A,v1500,z10,VentosaTCP\WObj:=PLACA_A;
    ENDPROC
    PROC Path_PSM2_A()
        MoveAbsJ PSM2_A,v1500,z10,VentosaTCP\WObj:=PLACA_A;
        MoveAbsJ PSM2_AA,v1500,z10,VentosaTCP\WObj:=PLACA_A;
        MoveAbsJ MID_A,v1500,z10,VentosaTCP\WObj:=PLACA_A;
        MoveAbsJ HOME_A,v1500,z10,VentosaTCP\WObj:=PLACA_A;
        MoveAbsJ MID_CONV_A,v1500,z10,VentosaTCP\WObj:=PLACA_A;
        MoveAbsJ CONVEYOR_A,v1500,z10,VentosaTCP\WObj:=PLACA_A;
    ENDPROC
    PROC Path_PSM2_AA()
        MoveAbsJ PSM2_AA,v1500,z10,VentosaTCP\WObj:=PLACA_A;
    ENDPROC
    PROC Path_SLIM2_AA()
        MoveAbsJ SLIM2_AA,v1500,z10,VentosaTCP\WObj:=PLACA_A;
    ENDPROC
    PROC Path_SLIM2_A()
        MoveAbsJ SLIM2_A,v1500,z10,VentosaTCP\WObj:=PLACA_A;
        MoveAbsJ SLIM2_AA,v1500,z10,VentosaTCP\WObj:=PLACA_A;
        MoveAbsJ MID_A,v1500,z10,VentosaTCP\WObj:=PLACA_A;
        MoveAbsJ HOME_A,v1500,z10,VentosaTCP\WObj:=PLACA_A;
        MoveAbsJ MID_CONV_A,v1500,z10,VentosaTCP\WObj:=PLACA_A;
        MoveAbsJ CONVEYOR_A,v1500,z10,VentosaTCP\WObj:=PLACA_A;
    ENDPROC
    PROC Path_SLDM2_AA()
        MoveAbsJ SLDM2_AA,v1500,z10,VentosaTCP\WObj:=PLACA_A;
    ENDPROC
    PROC Path_SLDM2_A()
        MoveAbsJ SLDM2_A,v1500,z10,VentosaTCP\WObj:=PLACA_A;
        MoveAbsJ SLDM2_AA,v1500,z10,VentosaTCP\WObj:=PLACA_A;
        MoveAbsJ MID_A,v1500,z10,VentosaTCP\WObj:=PLACA_A;
        MoveAbsJ HOME_A,v1500,z10,VentosaTCP\WObj:=PLACA_A;
        MoveAbsJ MID_CONV_A,v1500,z10,VentosaTCP\WObj:=PLACA_A;
        MoveAbsJ CONVEYOR_A,v1500,z10,VentosaTCP\WObj:=PLACA_A;
    ENDPROC

ENDMODULE

--- Backups/IRB1600APM/RAPID/TASK2/PROGMOD/CalibData.mod ---
MODULE CalibData
	PERS tooldata MyTool:=[TRUE,[[31.792631019,0,229.638935148],[0.945518576,0,0.325568154,0]],[1,[0,0,1],[1,0,0,0],0,0,0]];
	TASK PERS wobjdata PLACA_B:=[FALSE,TRUE,"",[[0,0,0],[1,0,0,0]],[[203.5,2358,-10],[0.707106781,0,0,-0.707106781]]];
ENDMODULE

--- Backups/IRB1600APM/RAPID/TASK2/PROGMOD/Module1.mod ---
MODULE Module1
	CONST jointtarget HOME_B:=[[0,0,0,0,30,0],[925,9E+09,9E+09,9E+09,9E+09,9E+09]];
	CONST jointtarget MID_B:=[[90,60,-20,0,50,0],[925,9E+09,9E+09,9E+09,9E+09,9E+09]];
    !***********************************************************
    !
    ! Módulo:  Module1
    !
    ! Descripción:
    !   <Introduzca la descripción aquí>
    !
    ! Autor: sebas
    !
    ! Versión: 1.0
    !
    !***********************************************************


    !***********************************************************
    !
    ! Procedimiento Main
    !
    !   Este es el punto de entrada de su programa
    !
    !***********************************************************
    PROC main()
        !Añada aquí su código
        Path_HOME_B;
        Path_MID_B;
        Path_HOME_B;
    ENDPROC
	PROC Path_HOME_B()
	    MoveAbsJ HOME_B,v1000,z100,MyTool\WObj:=PLACA_B;
	ENDPROC
	PROC Path_MID_B()
	    MoveAbsJ MID_B,v1000,z100,MyTool\WObj:=PLACA_B;
	ENDPROC
ENDMODULE

--- Backups/IRB1600APM/SYSPAR/EIO.cfg ---
EIO:CFG_1.0:6:1::
#
EIO_SIGNAL:

      -Name "START" -SignalType "DI" -Access "All"

      -Name "ATTACH" -SignalType "DO" -Access "All"

      -Name "MoveConv" -SignalType "DO" -Access "All"

      -Name "DRILLCHECK" -SignalType "DI" -Access "All"

      -Name "PAUSE" -SignalType "DO" -Access "All"

      -Name "DONE" -SignalType "DO" -Access "All"

      -Name "STOPDI" -SignalType "DI" -Access "All"
